TYPE "mlg2proPdi"
TITLE = {"version":"v1.0","author":"cyanezf","family":"core/dad/sick/mlg2","status":"current","deprecatedBy":null,"dependencies":[]}

//(*--
//# Documentation
//## Log
//| version | date | author | description |
//|:-------:|:----:|:------:|:------------|
//| v1.0 | 2026-08-31 | cyanezf | First version |
//
//## Description
//MLG2 barried PDI
//--*)
   STRUCT
      status : Struct   // 0.0: Status
         q1 : Bool;   // 0.0: Output status - Q1
         q2 : Bool;   // 0.1: Output status - Q2
         q3 : Bool;   // 0.2: Output status - Q3
         q4 : Bool;   // 0.3: Output status - Q4
         notUsed4 : Bool;   // 0.4
         notUsed5 : Bool;   // 0.5
         notUsed6 : Bool;   // 0.6
         notUsed7 : Bool;   // 0.7
         Qshortcircuit : Bool;   // 1.0: System status - 1=Q shortcircuit
         processDataInvalid : Bool;   // 1.1: System status - 1=Process data invalid
         overtemperature : Bool;   // 1.2: System status - 1=Overtemperature
         teachActive : Bool;   // 1.3: System status - 1=Teach active
         contaminationAlarm : Bool;   // 1.4: System status - 1=Contamination alarm
         hardwareError : Bool;   // 1.5: System status - 1=Hardware error
         teachFail : Bool;   // 1.6: System status - 1=Teach fail
         syncError : Bool;   // 1.7: System status - 1=Synchronization error
      END_STRUCT;
      data : Array[0..239] of Bool;   // 2.0: Data
   END_STRUCT;

END_TYPE

